Yaskawa INFORM job: R2-HOME.JBI

/JOB
//NAME R2-HOME
///FOLDERNAME FOLDER001
//POS
///NPOS 1,1,0,0,0,0
///TOOL 0
///POSTYPE ROBOT
///RECTAN
///RCONF 0,0,0,0,0,0,0,0,0,0,0,0,0,0,0,0,0,0,0,0,0,0,0,0
C00000=1043.307,21.310,-685.475,-3.2769,-33.1509,3.6066
BC00000=539.760,5648.937,840.904
//INST
///DATE 2023/07/10 17:09
///ATTR SC,RW,RJ
////FRAME ROBOT
///GROUP1 RB1,BS1
NOP
MOVJ C00000 BC00000 VJ=30.00
END
